{region '#Template'}
	{attribute 'Version' := '5.0.3.0'}
	{attribute 'Tags' := '"LCID": "1031", "Text": "Gebäudeautomation, Wetterstation, Thies"'}
	{attribute 'Tags' := '"LCID": "1033", "Text": "Building automation, Weatherstation, Thies"'}
	{attribute 'Using' := '"Type": "Template", "URI": "Site"'}
	{attribute 'Using' := '"Type": "Template", "URI": "BA2_Param"'}
	{attribute 'Using' := '"Type": "Template", "URI": "EC_ID"'}
	{attribute 'Using' := '"Type": "Template", "URI": "LblComp"'}		 
	{attribute 'Description' := '"LCID": "1031", "Text": "Haupt-Template mit schneller Task zum Lesen der seriellen Schnittstelle"'}
	{attribute 'Description' := '"LCID": "1033", "Text": "Main-template with fast task to read the serial Data from the terminal"'}
{endregion}
FUNCTION_BLOCK FB_BA_WeatherStation_Thies EXTENDS FB_BA_View
VAR_INPUT CONSTANT
	SerialCommRst				: FB_BA_Bv_OP;
	WthStRst					: FB_BA_Bv_OP;
	SerialCommErr				: FB_BA_BV;
	Dstb						: FB_BA_BV;
	Rain						: FB_BA_BI;
	WthT						: FB_BA_AI;
	DewPtT						: FB_BA_AI; 
	PrssAbs						: FB_BA_AI;
	PrssRel						: FB_BA_AI;
	HumAbs						: FB_BA_AI;
	HumRel						: FB_BA_AI;
	Brightness_N				: FB_BA_AI;
	Brightness_S				: FB_BA_AI;
	Brightness_E				: FB_BA_AI;
	Brightness_W				: FB_BA_AI;
	Dawn						: FB_BA_AI;
	GlobRadn					: FB_BA_AI;      
	WndDir						: FB_BA_AI;
	WndSpd						: FB_BA_AI; 
	Latd						: FB_BA_AI;  
	Lngt						: FB_BA_AI; 
	SunAzm						: FB_BA_AI;
	SunElv						: FB_BA_AI;                
END_VAR	

VAR
	ThiesWSC11					: FB_BA_ThiesWSC11;
	bResetWeatherStation		: BOOL;
	bResetSerialCommunication	: BOOL;
	DataConversion				: FB_BA_ThiesData;
	tonSerialCommErr			: TON;
	tonDstb						: TON;

	stRawDataIn			AT %I*	: KL6InData22B;	
	stRawDataOut 		AT %Q*	: KL6OutData22B;	
	fbSerialCtrl				: SerialLineControl;
	fbKL6Configuration			: KL6configuration;
	stTxBuff   					: ComBuffer;
	stRxBuff   					: ComBuffer;

	bSerialConfigError			: BOOL;
	nSerialConfigErrorID		: UDINT;
	bSerialCommError			: BOOL;
	nSerialCommErrorID			: UDINT;
	
	bAccumulatedSerialError		: BOOL;
	bAccumulatedDisturbance		: BOOL;
END_VAR                 

VAR_INPUT CONSTANT PERSISTENT
	{attribute 'parameterUnit':= 's'}
	nSerialCommErrDelay 		: UDINT := 10;
	{attribute 'parameterUnit':= 's'}
	nDstbDelay 					: UDINT := 10;
END_VAR
VAR // added by the converter: edge detectors and wires of the graphical bodies
    _w1 : BOOL;
    _w2, _w3, _w4 : ANY;
END_VAR

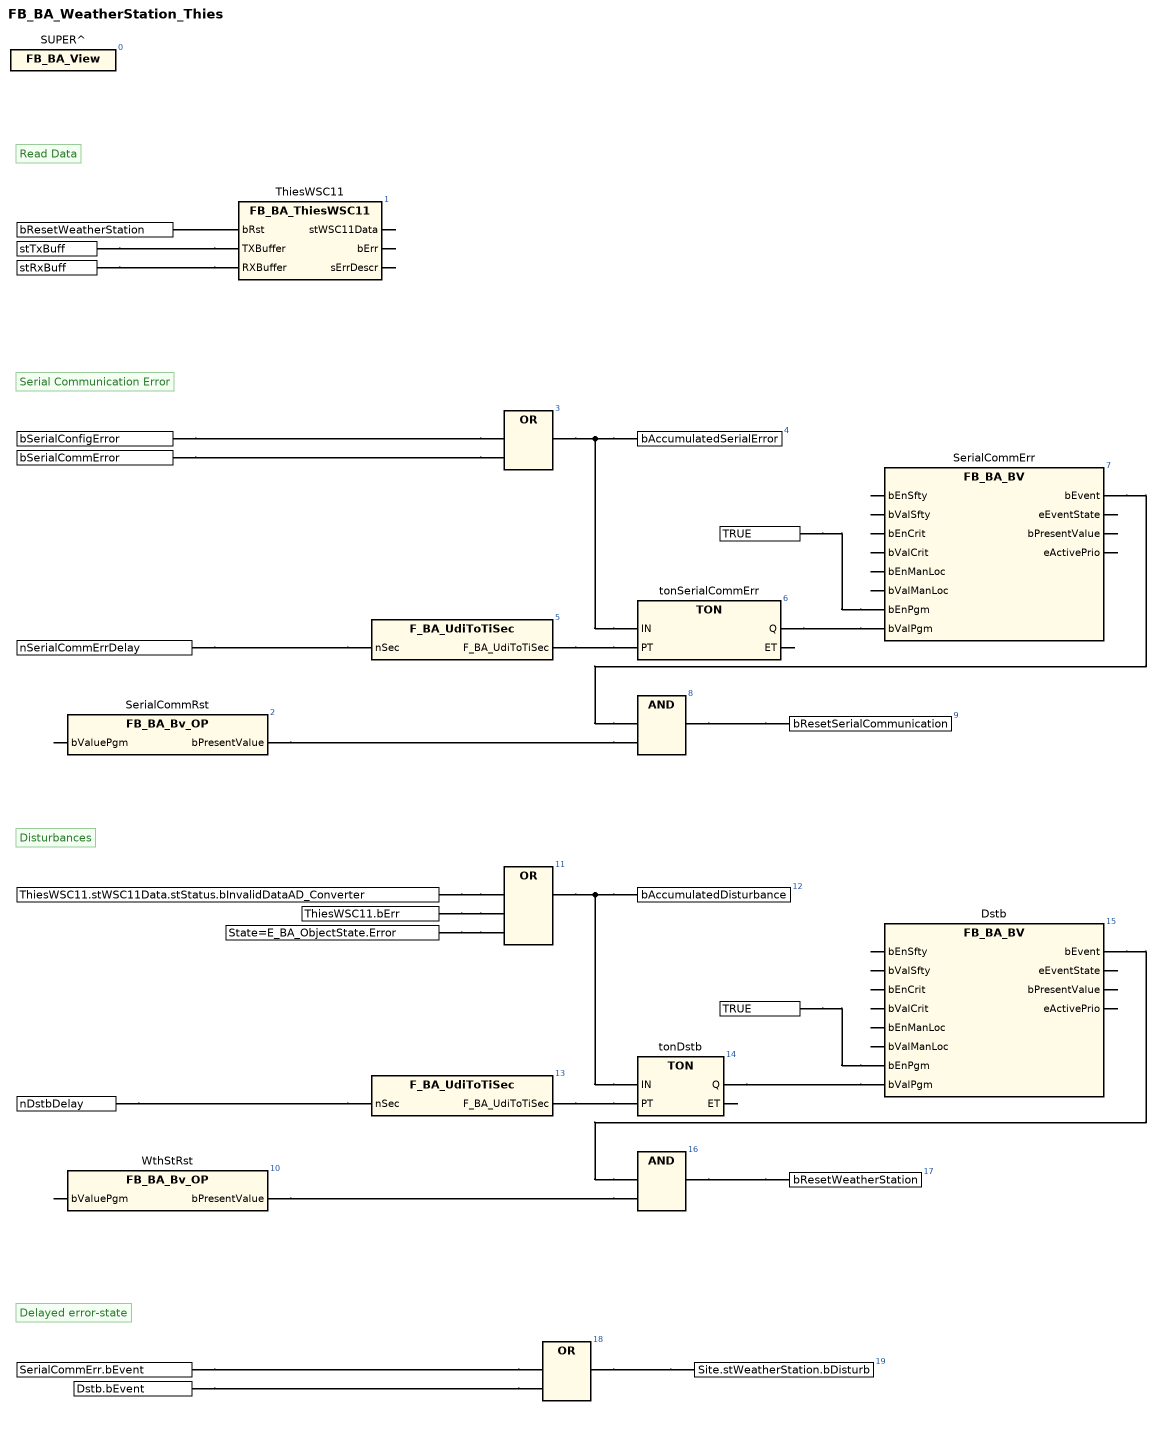
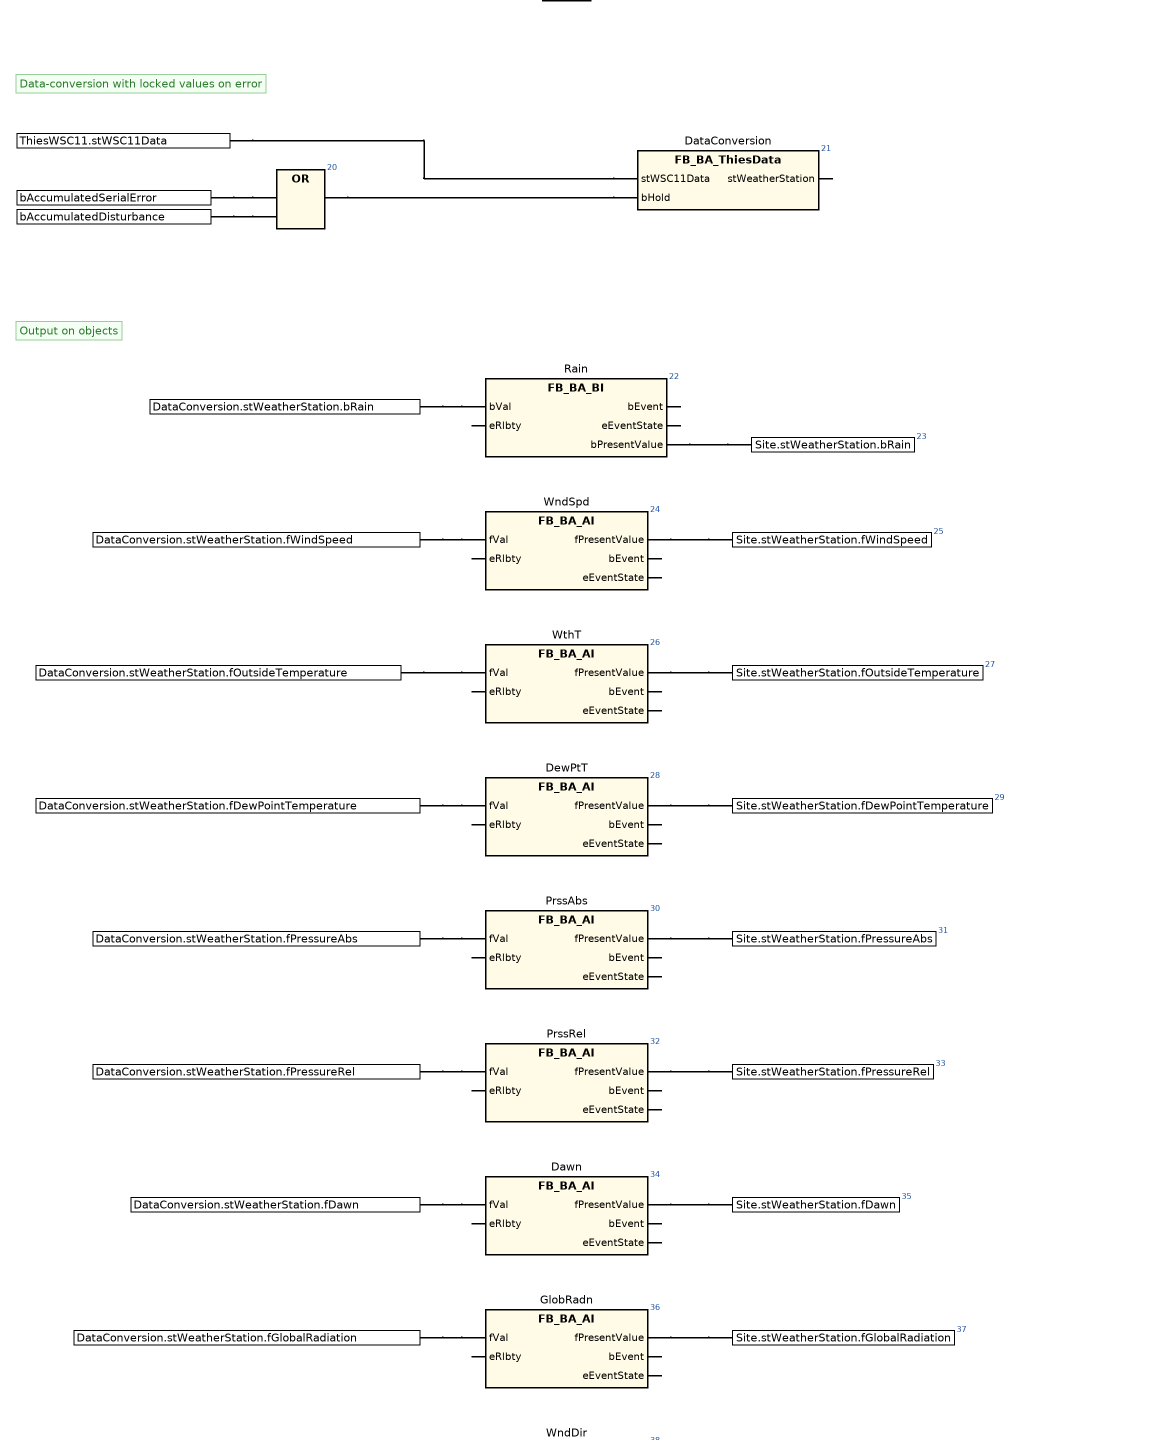
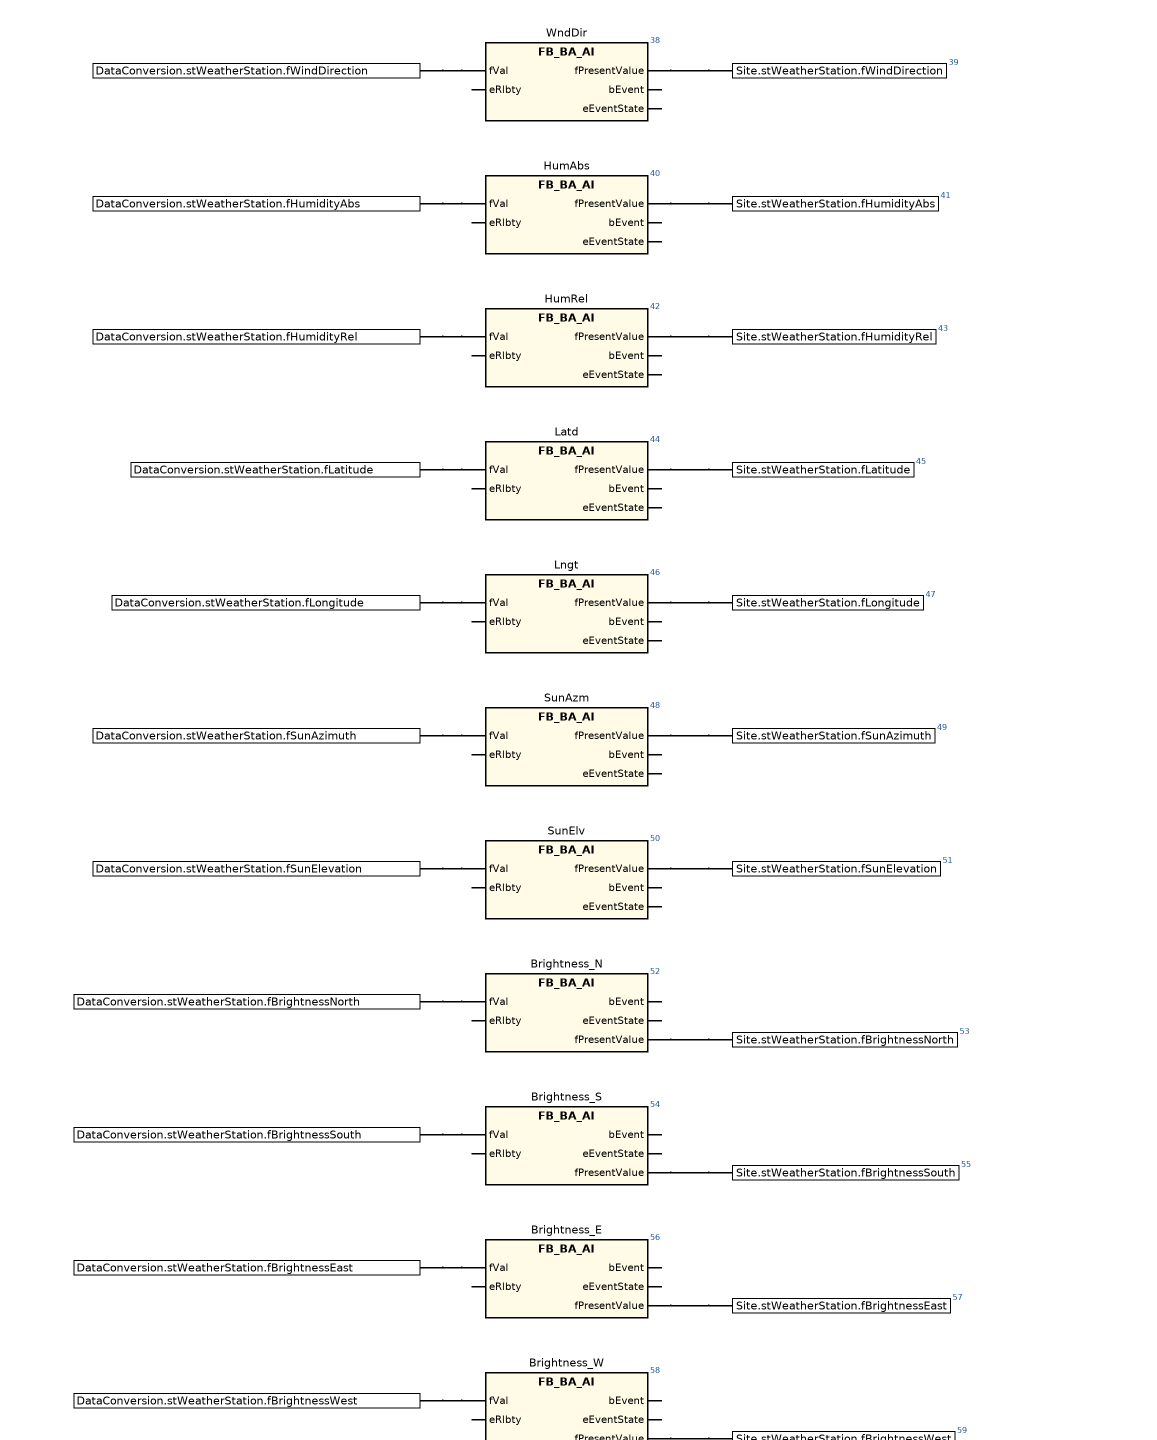
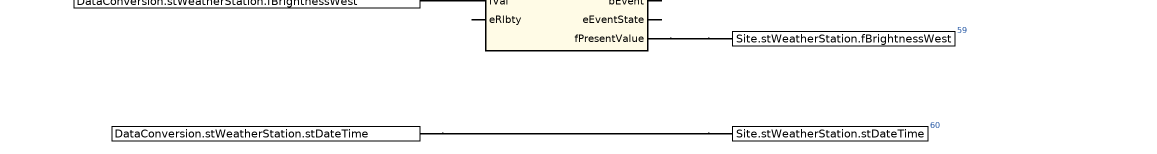
SUPER^(); // FB_BA_View
// Read Data
ThiesWSC11(bRst := bResetWeatherStation, TXBuffer := stTxBuff, RXBuffer := stRxBuff); // FB_BA_ThiesWSC11
SerialCommRst(); // FB_BA_Bv_OP
// Serial Communication Error
_w1 := bSerialConfigError OR bSerialCommError;
bAccumulatedSerialError := _w1;
_w2 := F_BA_UdiToTiSec(nSec := nSerialCommErrDelay);
tonSerialCommErr(IN := _w1, PT := _w2); // TON
SerialCommErr(bEnPgm := TRUE, bValPgm := tonSerialCommErr.Q); // FB_BA_BV
bResetSerialCommunication := SerialCommErr.bEvent AND SerialCommRst.bPresentValue;
WthStRst(); // FB_BA_Bv_OP
// Disturbances
_w3 := ThiesWSC11.stWSC11Data.stStatus.bInvalidDataAD_Converter OR ThiesWSC11.bErr OR (State=E_BA_ObjectState.Error);
bAccumulatedDisturbance := _w3;
_w4 := F_BA_UdiToTiSec(nSec := nDstbDelay);
tonDstb(IN := _w3, PT := _w4); // TON
Dstb(bEnPgm := TRUE, bValPgm := tonDstb.Q); // FB_BA_BV
bResetWeatherStation := Dstb.bEvent AND WthStRst.bPresentValue;
// Delayed error-state
Site.stWeatherStation.bDisturb := SerialCommErr.bEvent OR Dstb.bEvent;
// Data-conversion with locked values on error
DataConversion(stWSC11Data := ThiesWSC11.stWSC11Data, bHold := bAccumulatedSerialError OR bAccumulatedDisturbance); // FB_BA_ThiesData
// Output on objects
Rain(bVal := DataConversion.stWeatherStation.bRain); // FB_BA_BI
Site.stWeatherStation.bRain := Rain.bPresentValue;
WndSpd(fVal := DataConversion.stWeatherStation.fWindSpeed); // FB_BA_AI
Site.stWeatherStation.fWindSpeed := WndSpd.fPresentValue;
WthT(fVal := DataConversion.stWeatherStation.fOutsideTemperature); // FB_BA_AI
Site.stWeatherStation.fOutsideTemperature := WthT.fPresentValue;
DewPtT(fVal := DataConversion.stWeatherStation.fDewPointTemperature); // FB_BA_AI
Site.stWeatherStation.fDewPointTemperature := DewPtT.fPresentValue;
PrssAbs(fVal := DataConversion.stWeatherStation.fPressureAbs); // FB_BA_AI
Site.stWeatherStation.fPressureAbs := PrssAbs.fPresentValue;
PrssRel(fVal := DataConversion.stWeatherStation.fPressureRel); // FB_BA_AI
Site.stWeatherStation.fPressureRel := PrssRel.fPresentValue;
Dawn(fVal := DataConversion.stWeatherStation.fDawn); // FB_BA_AI
Site.stWeatherStation.fDawn := Dawn.fPresentValue;
GlobRadn(fVal := DataConversion.stWeatherStation.fGlobalRadiation); // FB_BA_AI
Site.stWeatherStation.fGlobalRadiation := GlobRadn.fPresentValue;
WndDir(fVal := DataConversion.stWeatherStation.fWindDirection); // FB_BA_AI
Site.stWeatherStation.fWindDirection := WndDir.fPresentValue;
HumAbs(fVal := DataConversion.stWeatherStation.fHumidityAbs); // FB_BA_AI
Site.stWeatherStation.fHumidityAbs := HumAbs.fPresentValue;
HumRel(fVal := DataConversion.stWeatherStation.fHumidityRel); // FB_BA_AI
Site.stWeatherStation.fHumidityRel := HumRel.fPresentValue;
Latd(fVal := DataConversion.stWeatherStation.fLatitude); // FB_BA_AI
Site.stWeatherStation.fLatitude := Latd.fPresentValue;
Lngt(fVal := DataConversion.stWeatherStation.fLongitude); // FB_BA_AI
Site.stWeatherStation.fLongitude := Lngt.fPresentValue;
SunAzm(fVal := DataConversion.stWeatherStation.fSunAzimuth); // FB_BA_AI
Site.stWeatherStation.fSunAzimuth := SunAzm.fPresentValue;
SunElv(fVal := DataConversion.stWeatherStation.fSunElevation); // FB_BA_AI
Site.stWeatherStation.fSunElevation := SunElv.fPresentValue;
Brightness_N(fVal := DataConversion.stWeatherStation.fBrightnessNorth); // FB_BA_AI
Site.stWeatherStation.fBrightnessNorth := Brightness_N.fPresentValue;
Brightness_S(fVal := DataConversion.stWeatherStation.fBrightnessSouth); // FB_BA_AI
Site.stWeatherStation.fBrightnessSouth := Brightness_S.fPresentValue;
Brightness_E(fVal := DataConversion.stWeatherStation.fBrightnessEast); // FB_BA_AI
Site.stWeatherStation.fBrightnessEast := Brightness_E.fPresentValue;
Brightness_W(fVal := DataConversion.stWeatherStation.fBrightnessWest); // FB_BA_AI
Site.stWeatherStation.fBrightnessWest := Brightness_W.fPresentValue;
Site.stWeatherStation.stDateTime := DataConversion.stWeatherStation.stDateTime;

METHOD FastCycle

VAR_INST
	nStepSerialComm			: INT;
	rtReset					: R_TRIG;
	nConfigErrorCounter		: USINT;
	tonWait					: TON;
END_VAR
rtReset(CLK:=bResetSerialCommunication);


CASE	nStepSerialComm	OF
	0:	//idle
		nStepSerialComm	:= 10;
	
	10: //init
		fbKL6Configuration(
			Execute := TRUE,
			Mode := SERIALLINEMODE_KL6_22B_STANDARD,
			Baudrate := 9600,
			NoDatabits := 8,
			Parity := PARITY_NONE,
			Stopbits := 1,
			Handshake := RS485_HALFDUPLEX,
			ContinousMode := FALSE,
			pComIn := ADR(stRawDataIn),
			pComOut := ADR(stRawDataOut),
			SizeComIn := SIZEOF(stRawDataIn)
		);
		
		IF (NOT fbKL6Configuration.Busy) THEN
			fbKL6Configuration(	Execute := FALSE);
			IF fbKL6Configuration.Error	THEN
				nStepSerialComm	:= 20;
			ELSE	
				nStepSerialComm	:= 50;
			END_IF
		END_IF
	
	20:	// error-counter
		nConfigErrorCounter	:= nConfigErrorCounter+1;
		IF nConfigErrorCounter > 5	THEN
			nStepSerialComm	:= 40;
		ELSE 
			nStepSerialComm	:= 30;
		END_IF
		
	30:	// wait restart config
		tonWait(IN:=TRUE, PT:=T#5S);	
		IF tonWait.Q				THEN	
			tonWait(IN:=FALSE);
			nStepSerialComm	:= 10;
		END_IF
		
	40: // configuration error	
		bSerialConfigError	:= TRUE;
		IF rtReset.Q	THEN
			bSerialConfigError	:= FALSE;
			nConfigErrorCounter	:= 0;
			nStepSerialComm		:= 10;
		END_IF
		
	50: // run communication	
		fbSerialCtrl(
			Mode		:= SERIALLINEMODE_KL6_22B_STANDARD,
			pComIn		:= ADR(stRawDataIn),
			pComOut		:= ADR(stRawDataOut),
			SizeComIn	:= TO_INT(SIZEOF(stRawDataIn)),
			TxBuffer	:= stTxBuff,
			RxBuffer	:= stRxBuff,
		);
		
		tonWait(IN:=fbSerialCtrl.Error, PT:=T#10S);
		IF tonWait.Q	THEN
				tonWait(IN:=FALSE);
				nStepSerialComm	:= 60;
		END_IF
		
	60: // communication error	
		bSerialCommError	:= TRUE;
		IF rtReset.Q	THEN
			bSerialCommError	:= FALSE;
			nStepSerialComm		:= 50;
		END_IF
END_CASE

nSerialConfigErrorID	:= TO_UDINT(fbKL6Configuration.ErrorID);
nSerialCommErrorID		:= TO_UDINT(fbSerialCtrl.ErrorID);
END_METHOD

METHOD FB_init : BOOL
VAR_INPUT
	bInitRetains : BOOL; // if TRUE, the retain variables are initialized (warm start / cold start)
	bInCopyCode : BOOL;  // if TRUE, the instance afterwards gets moved into the copy code (online change)
END_VAR
ThiesWSC11.nUpdateTime					:= 500; 		// data-polling interval [500..60000ms]
ThiesWSC11.nWndDatAvrgIntVal			:= 0;			// Wind data averaging intervall - 0 = Off; 1-10 = minutes
ThiesWSC11.bTwiLgtCalcAvrg				:= FALSE;		// Twilight-caluclation average - FALSE = Sum of the light-sensors is taken ; TRUE = Average of the light-sensors is taken 		
ThiesWSC11.nWndDirNorthOffs				:= 0;			// Wind direction North offset (correction) [0..360°]
ThiesWSC11.nStHgtAMSL					:= 0;			// Station height above mean sea level [0..3000m], 3001 means, that the level is automatically taken from GPS-device
ThiesWSC11.nRainOffDly					:= 0;			// Rain off delay [0..3600s]	
ThiesWSC11.nDistMsgDly					:= 0;			// Disturbance message delay [0..60s]
										
										
SerialCommRst.iParent					:= THIS^;
SerialCommRst.iLabel					:= LblComp_Wth_WeatherStationCommReset; 	
SerialCommRst.sInactiveText				:= txtEvent_Off;
SerialCommRst.sActiveText				:= txtEvent_On;
SerialCommRst.bValueRm					:= FALSE;
SerialCommRst.eToggleMode				:= E_BA_ToggleMode.ePushButton;    
										
WthStRst.iParent						:= THIS^;
WthStRst.iLabel							:= LblComp_Wth_WeatherStationReset; 
WthStRst.sInactiveText					:= txtEvent_Off;
WthStRst.sActiveText					:= txtEvent_On;
WthStRst.bValueRm						:= FALSE;
WthStRst.eToggleMode					:= E_BA_ToggleMode.ePushButton;  
                                        
SerialCommErr.iParent					:= THIS^;
SerialCommErr.iLabel					:= LblComp_Wth_WeatherStationComm; 
SerialCommErr.sActiveText 				:= txtEvent_Triggered;
SerialCommErr.sInactiveText 			:= txtEvent_Normal;
SerialCommErr.bEnManualRm				:= FALSE;	//	Priority  8	
SerialCommErr.bValManualRm				:= FALSE;	//	Priority  8
SerialCommErr.nEventClassID				:= EC_ID.NC30;
SerialCommErr.stTimeDelay.nToNormal		:= 0;
SerialCommErr.stTimeDelay.nToAbnormal	:= 0;
SerialCommErr.bAlarmValue				:= TRUE;
SerialCommErr.aEventTransitionText[1]	:= txtEvent_Triggered;
SerialCommErr.aEventTransitionText[2]	:= txtEvent_Error;
SerialCommErr.aEventTransitionText[3]	:= txtEvent_Normal;
SerialCommErr.bEventDetectionEnable		:= TRUE;
SerialCommErr.eEnPlantLock				:= E_BA_LockPriority.eNoLock;
                                        
Dstb.iParent							:= THIS^;
Dstb.iLabel								:= LblComp_Wth_WeatherStation;   	
Dstb.sActiveText 						:= txtEvent_Triggered;
Dstb.sInactiveText 						:= txtEvent_Normal;
Dstb.bEnManualRm						:= FALSE;	//	Priority  8	
Dstb.bValManualRm						:= FALSE;	//	Priority  8
Dstb.nEventClassID						:= EC_ID.NC30;
Dstb.stTimeDelay.nToNormal				:= 0;
Dstb.stTimeDelay.nToAbnormal			:= 0;
Dstb.bAlarmValue						:= TRUE;
Dstb.aEventTransitionText[1]			:= txtEvent_Triggered;
Dstb.aEventTransitionText[2]			:= txtEvent_Error;
Dstb.aEventTransitionText[3]			:= txtEvent_Normal;
Dstb.bEventDetectionEnable				:= TRUE;
Dstb.eEnPlantLock						:= E_BA_LockPriority.eNoLock;
												
Rain.iParent							:= THIS^;
Rain.iLabel								:= LblComp_Wth_RainSensor; 	
Rain.sActiveText 						:= txtEvent_Yes;
Rain.sInactiveText 						:= txtEvent_No;
Rain.nEventClassID						:= EC_ID.NC60;
Rain.aEventTransitionText[1]			:= txtEvent_No;
Rain.aEventTransitionText[2]			:= txtEvent_None;
Rain.aEventTransitionText[3]			:= txtEvent_Yes;
Rain.bEventDetectionEnable				:= FALSE;	
						
WthT.iParent							:= THIS^;
WthT.iLabel								:= LblComp_Wth_TemperatureOutside; 	
WthT.eUnit 								:= E_BA_Unit.eTemperature_DegreesCelsius;	
WthT.nEventClassID						:= EC_ID.NC40;

										
DewPtT.iParent							:= THIS^;
DewPtT.iLabel							:= LblComp_Wth_TemperatureDewPoint; 		
DewPtT.eUnit							:= E_BA_Unit.eTemperature_DegreesCelsius;
DewPtT.nEventClassID					:= EC_ID.NC40;
						
PrssAbs.iParent							:= THIS^;
PrssAbs.iLabel							:= LblComp_Wth_PressureAbsolute; 
PrssAbs.eUnit							:= E_BA_Unit.ePressure_Hectopascals;
PrssAbs.nEventClassID					:= EC_ID.NC40;

										
PrssRel.iParent							:= THIS^;
PrssRel.iLabel							:= LblComp_Wth_PressureRelative; 	
PrssRel.eUnit							:= E_BA_Unit.ePressure_Hectopascals;
PrssRel.nEventClassID					:= EC_ID.NC40;
						
HumAbs.iParent							:= THIS^;
HumAbs.iLabel							:= LblComp_Wth_AbsoluteHumidityOutsideAir; 
HumAbs.eUnit							:= E_BA_Unit.eHumidity_GramsOfWaterPerKilogramDryAir;
HumAbs.nEventClassID					:= EC_ID.NC40;
										
HumRel.iParent							:= THIS^;
HumRel.iLabel							:= LblComp_Wth_RelativeHumidityOutsideAir; 
HumRel.eUnit							:= E_BA_Unit.eHumidity_PercentRelativeHumidity;
HumRel.nEventClassID					:= EC_ID.NC40;
						
Brightness_N.iParent					:= THIS^;
Brightness_N.iLabel						:= LblComp_Wth_Brightness; 		
Brightness_N.eUnit						:= E_BA_Unit.eLight_Luxes;
Brightness_N.nEventClassID				:= EC_ID.NC40;
                                        
Brightness_S.iParent					:= THIS^;
Brightness_S.iLabel						:= LblComp_Wth_Brightness; 		
Brightness_S.eUnit						:= E_BA_Unit.eLight_Luxes;
Brightness_S.nEventClassID				:= EC_ID.NC40;
                                        
Brightness_E.iParent					:= THIS^;
Brightness_E.iLabel						:= LblComp_Wth_Brightness; 		
Brightness_E.eUnit						:= E_BA_Unit.eLight_Luxes;
Brightness_E.nEventClassID				:= EC_ID.NC40;
                                        
Brightness_W.iParent					:= THIS^;
Brightness_W.iLabel						:= LblComp_Wth_Brightness; 		
Brightness_W.eUnit						:= E_BA_Unit.eLight_Luxes;
Brightness_W.nEventClassID				:= EC_ID.NC40;

Dawn.iParent							:= THIS^;
Dawn.iLabel								:= LblComp_Wth_Dawn; 	
Dawn.eUnit								:= E_BA_Unit.eLight_Luxes;
Dawn.nEventClassID						:= EC_ID.NC40;
						
GlobRadn.iParent						:= THIS^;
GlobRadn.iLabel							:= LblComp_Wth_SolarRadiation; 	
GlobRadn.eUnit							:= E_BA_Unit.eLight_WattsPerSquareMeter;
GlobRadn.nEventClassID					:= EC_ID.NC40;
						
WndDir.iParent							:= THIS^;
WndDir.iLabel							:= LblComp_Wth_WindDirection; 	
WndDir.eUnit							:= E_BA_Unit.eOther_DegreesAngular;
WndDir.nEventClassID					:= EC_ID.NC40;
										
WndSpd.iParent							:= THIS^;
WndSpd.iLabel							:= LblComp_Wth_WindSpeed; 	
WndSpd.eUnit							:= E_BA_Unit.eVelocity_MetersPerSecond;
WndSpd.nEventClassID					:= EC_ID.NC40;
						
Latd.iParent							:= THIS^;
Latd.iLabel								:= LblComp_Wth_GeoLatitude; 	
Latd.eUnit								:= E_BA_Unit.eOther_DegreesAngular;
Latd.nEventClassID						:= EC_ID.NC40;
										
Lngt.iParent							:= THIS^;
Lngt.iLabel								:= LblComp_Wth_GeoLongitude; 	
Lngt.eUnit								:= E_BA_Unit.eOther_DegreesAngular;
Lngt.nEventClassID						:= EC_ID.NC40;
						
SunAzm.iParent							:= THIS^;
SunAzm.iLabel							:= LblComp_Wth_SunAzimuth; 	
SunAzm.eUnit							:= E_BA_Unit.eOther_DegreesAngular;
SunAzm.nEventClassID					:= EC_ID.NC40;
						
SunElv.iParent							:= THIS^;
SunElv.iLabel							:= LblComp_Wth_SunElevation; 	
SunElv.eUnit							:= E_BA_Unit.eOther_DegreesAngular;
SunElv.nEventClassID					:= EC_ID.NC40;
END_METHOD

END_FUNCTION_BLOCK

(* stored: Version 1.1.0.1, ProductVersion 3.1.4024.12
   POU FB_BA_WeatherStation_Thies: Id {46291e31-f6f5-41a8-8f1b-90c9c9ab208d}, SpecialFunc None
   Folder Fast Task: Id {6aab4a21-52e1-4a42-86ac-f9648a9882c5}
   Method FastCycle: Id {3479beb4-4093-47a6-89a9-652da1379f6b}
   Method FB_init: Id {248253f5-e0c7-4bc0-ac8d-94f6300566f6} *)
